ABB RobotStudio station: simulacion_final.rspag

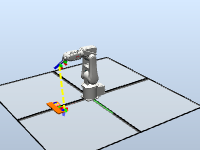
--- station ---
Station funciona (saved by RobotStudio 6.8.8307.1040)
Controller Sistema3
  mechanical unit ROB_1: IRB120_3_58__01, 6 joints, base frame (0, 0, 0) mm
Layout (positions relative to the parent item):
  - IRB120_3_58__01 [mechanism, from Robots\IRB120_3_58_G_01.rslib] at (0, 0, 0) mm; joint values [0, 0, 0, 0, 0.5236, 0] (rad or m)
  - PIANO [part] at (456.26, 0.5, 5) mm, rotated rx 180 ry 0 rz 0 deg
  - Herramienta [mechanism] at (364.35, 0, 594) mm, rotated rx 180 ry 60 rz 180 deg
      TCP Herramienta at (0, 0, 68.75) mm
      links: HERRAMIENTA
  - PIANO [part]
Attachment: Herramienta is attached to IRB120_3_58__01 / Link6

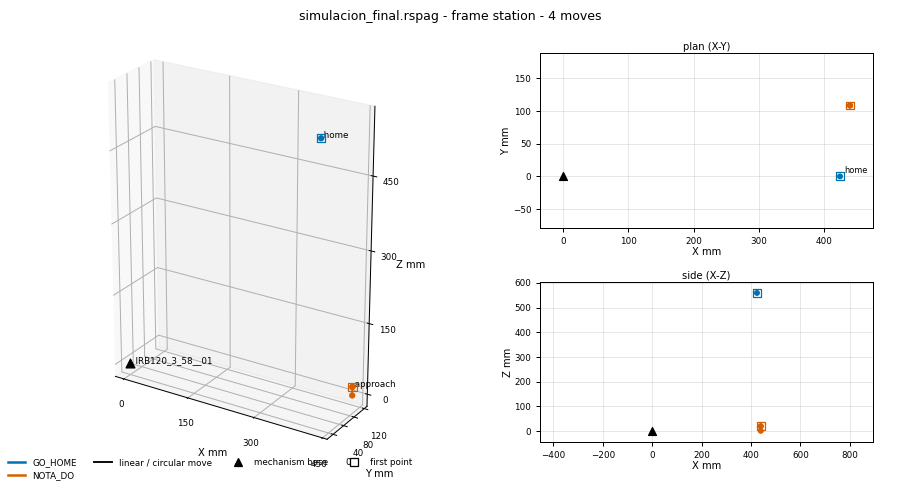
[picture p0: tool path of simulacion_final.rspag in frame station, 4 of 25 moves have a stored position in this frame; points joined in program order, loops and branches not executed]
--- Backups/Sistema3/RAPID/TASK1/PROGMOD/CalibData.mod ---
MODULE CalibData
	PERS tooldata Herramienta:=[TRUE,[[0,0,68.75],[1,0,0,0]],[1,[0,0,1],[1,0,0,0],0,0,0]];
ENDMODULE

--- Backups/Sistema3/RAPID/TASK1/PROGMOD/Module1.mod ---
MODULE Module1
    CONST robtarget home:=[[423.893075583,0,559.625],[0.5,0,0.866025404,0],[0,0,0,0],[9E+09,9E+09,9E+09,9E+09,9E+09,9E+09]];
    CONST robtarget approach:=[[439.246604644,108.499999249,20.160944941],[0.123487824,0.000000005,0.992346087,0.000000004],[0,-1,0,0],[9E+09,9E+09,9E+09,9E+09,9E+09,9E+09]];
    CONST robtarget pulse:=[[439.246586904,108.499996962,1.527563706],[0.123487794,0.000000019,0.992346091,0.000000006],[0,-1,0,0],[9E+09,9E+09,9E+09,9E+09,9E+09,9E+09]];

    ! separación entre teclas (mm)
    CONST num dist_tecla := 31;

    ! SOCKET ÚNICO
    VAR socketdev ServerSocket;
    VAR socketdev ClientSocket;

    ! Variables
    VAR bool ejecutar := TRUE;
    VAR string cmd;

PROC main()

    ! inicializar socket único
    SocketCreate ServerSocket;
    SocketBind ServerSocket, "127.0.0.1", 7000;
    SocketListen ServerSocket;

    !SocketSend ClientSocket, \str:="Conexión correcta";

    GO_HOME;

    WHILE ejecutar DO

        SocketAccept ServerSocket, ClientSocket, \Time:=WAIT_MAX;

        cmd := "";

        ! Recibe (se queda esperando datos en el socket que ya se cerró)
        SocketReceive ClientSocket, \str:=cmd\Time:=WAIT_MAX;

        ! quitar posible salto de línea final
        IF StrLen(cmd) > 0 THEN
            cmd := StrPart(cmd, 1, StrLen(cmd) - 1);
        ENDIF

        IF StrLen(cmd) = 0 THEN
            !ejecutar := FALSE;
            SocketSend ClientSocket, \str:="ERROR: VACIO";
            !EXIT;
        ELSEIF cmd = "QUIT" THEN
            ejecutar := FALSE;
            SocketSend ClientSocket, \str:="SALIENDO";
            !EXIT;
        ELSE
            TOCAR(cmd);
        ENDIF

        SocketClose ClientSocket;

    ENDWHILE

    GO_HOME;

    ! finalizar socket
    SocketClose ServerSocket;

ENDPROC

    PROC GO_HOME()
        MoveJ home, v200, fine, Herramienta\WObj:=wobj0;
    ENDPROC

    PROC TOCAR(string nota)

        IF nota = "D" THEN
            NOTA_DO;
            SocketSend ClientSocket, \str:="DO";
        ELSEIF nota = "R" THEN
            NOTA_RE;
            SocketSend ClientSocket, \str:="RE";
        ELSEIF nota = "M" THEN
            NOTA_MI;
            SocketSend ClientSocket, \str:="MI";
        ELSEIF nota = "F" THEN
            NOTA_FA;
            SocketSend ClientSocket, \str:="FA";
        ELSEIF nota = "S" THEN
            NOTA_SOL;
            SocketSend ClientSocket, \str:="SOL";
        ELSEIF nota = "L" THEN
            NOTA_LA;
            SocketSend ClientSocket, \str:="LA";
        ELSEIF nota = "I" THEN
            NOTA_SI;
            SocketSend ClientSocket, \str:="SI";
        ELSEIF nota = "O" THEN
            NOTA_DO_SOST;
            SocketSend ClientSocket, \str:="DO_SOST";
!        ELSEIF nota = "H" THEN
!            CUMPLEANYOS;
!            SocketSend ClientSocket, \str:="CUMPLE";
        ELSEIF nota = "H" THEN
            GO_HOME;
            SocketSend ClientSocket, \str:="HOME";
        ELSEIF nota = "1" THEN
            SocketSend ClientSocket, \str:="OK MODO";
        ELSEIF nota = "2" THEN
            SocketSend ClientSocket, \str:="OK MODO";
        ELSEIF nota = "3" THEN
            SocketSend ClientSocket, \str:="OK MODO";
        ELSEIF nota = "4" THEN
            SocketSend ClientSocket, \str:="OK MODO";
        ELSE
            SocketSend ClientSocket, \str:="ERROR";
        ENDIF

    ENDPROC

    PROC NOTA_DO()
        MoveJ approach, v200, z100, Herramienta\WObj:=wobj0;
        MoveL pulse,    v50,  fine, Herramienta\WObj:=wobj0;
        MoveL approach, v200, fine, Herramienta\WObj:=wobj0;
    ENDPROC

    PROC NOTA_RE()
        MoveJ Offs(approach, 0, -1*dist_tecla, 0), v200, z100, Herramienta\WObj:=wobj0;
        MoveL Offs(pulse,    0, -1*dist_tecla, 0), v50,  fine, Herramienta\WObj:=wobj0;
        MoveL Offs(approach, 0, -1*dist_tecla, 0), v200, fine, Herramienta\WObj:=wobj0;
    ENDPROC

    PROC NOTA_MI()
        MoveJ Offs(approach, 0, -2*dist_tecla, 0), v200, z100, Herramienta\WObj:=wobj0;
        MoveL Offs(pulse,    0, -2*dist_tecla, 0), v50,  fine, Herramienta\WObj:=wobj0;
        MoveL Offs(approach, 0, -2*dist_tecla, 0), v200, fine, Herramienta\WObj:=wobj0;
    ENDPROC

    PROC NOTA_FA()
        MoveJ Offs(approach, 0, -3*dist_tecla, 0), v200, z100, Herramienta\WObj:=wobj0;
        MoveL Offs(pulse,    0, -3*dist_tecla, 0), v50,  fine, Herramienta\WObj:=wobj0;
        MoveL Offs(approach, 0, -3*dist_tecla, 0), v200, fine, Herramienta\WObj:=wobj0;
    ENDPROC

    PROC NOTA_SOL()
        MoveJ Offs(approach, 0, -4*dist_tecla, 0), v200, z100, Herramienta\WObj:=wobj0;
        MoveL Offs(pulse,    0, -4*dist_tecla, 0), v50,  fine, Herramienta\WObj:=wobj0;
        MoveL Offs(approach, 0, -4*dist_tecla, 0), v200, fine, Herramienta\WObj:=wobj0;
    ENDPROC

    PROC NOTA_LA()
        MoveJ Offs(approach, 0, -5*dist_tecla, 0), v200, z100, Herramienta\WObj:=wobj0;
        MoveL Offs(pulse,    0, -5*dist_tecla, 0), v50,  fine, Herramienta\WObj:=wobj0;
        MoveL Offs(approach, 0, -5*dist_tecla, 0), v200, fine, Herramienta\WObj:=wobj0;
    ENDPROC

    PROC NOTA_SI()
        MoveJ Offs(approach, 0, -6*dist_tecla, 0), v200, z100, Herramienta\WObj:=wobj0;
        MoveL Offs(pulse,    0, -6*dist_tecla, 0), v50,  fine, Herramienta\WObj:=wobj0;
        MoveL Offs(approach, 0, -6*dist_tecla, 0), v200, fine, Herramienta\WObj:=wobj0;
    ENDPROC

    PROC NOTA_DO_SOST()
        MoveJ Offs(approach, 0, -7*dist_tecla, 0), v200, z100, Herramienta\WObj:=wobj0;
        MoveL Offs(pulse,    0, -7*dist_tecla, 0), v50,  fine, Herramienta\WObj:=wobj0;
        MoveL Offs(approach, 0, -7*dist_tecla, 0), v200, fine, Herramienta\WObj:=wobj0;
    ENDPROC

!    PROC CUMPLEANYOS()
!       ! DO DO RE DO FA MI        (Cum-ple-a-ños fe-liz)
!       ! DO DO RE DO SOL FA       (Cum-ple-a-ños fe-liz)
!       ! DO DO DO_SOST LA FA MI RE (Te de-se-a-mos to-dos)
!       ! SI SI LA FA SOL FA       (Cum-ple-a-ños fe-liz)

!        ! --- Línea 1 ---
!        NOTA_DO;
!        NOTA_DO;
!        NOTA_RE;
!        NOTA_DO;
!        NOTA_FA;
!        NOTA_MI;

!        ! --- Línea 2 ---
!        NOTA_DO;
!        NOTA_DO;
!        NOTA_RE;
!        NOTA_DO;
!        NOTA_SOL;
!        NOTA_FA;

!        ! --- Línea 3 ---
!        NOTA_DO;
!        NOTA_DO;
!        NOTA_DO_SOST;
!        NOTA_LA;
!        NOTA_FA;
!        NOTA_MI;
!        NOTA_RE;

!        ! --- Línea 4 ---
!        NOTA_SI;
!        NOTA_SI;
!        NOTA_LA;
!        NOTA_FA;
!        NOTA_SOL;
!        NOTA_FA;
!    ENDPROC

ENDMODULE
